// TwinCAT 3 PLC project Virtual_plc
// ProgramVersion: 3.1.4024.0
// libraries:
//   Tc2_Standard, * (Beckhoff Automation GmbH)
//   Tc2_System, * (Beckhoff Automation GmbH)
//   Tc3_Module, * (Beckhoff Automation GmbH)
// project tree:
//   GVLs/ GVL.TcGVL
//   / PlcTask.TcTTO, TASK_2.TcTTO
//   POUs/ Wait.TcPOU, Step.TcDUT, Task_1.TcPOU, Taks_2.TcPOU
// real-time tasks:
//   TASK PlcTask: cycle T#3000ms, priority 20, ADS port 350
//   TASK TASK 2: cycle T#1ms, priority 1, ADS port 351

CONFIGURATION Virtual_plc
    RESOURCE PLC ON TwinCAT3
        TASK PlcTask(INTERVAL := T#3000ms, PRIORITY := 20);
        TASK TASK_2(INTERVAL := T#1ms, PRIORITY := 1);
        PROGRAM Task_1 WITH PlcTask : Task_1;
        PROGRAM Taks_2 WITH TASK_2 : Taks_2;
    END_RESOURCE
END_CONFIGURATION

// ---- POUs/Step.TcDUT
TYPE Step :
//ALl the case steps
(
	sleeping, 
	alarm, 
	snooze1, 
	snooze2, 
	wake, 
	toilet1,
	kitchen, 
	breakfast, 
	lunch, 
	toilet2, 
	garage, 
	cycling,
	train_check, 
	done	
) := sleeping;
END_TYPE

// ---- GVLs/GVL.TcGVL
{attribute 'qualified_only'}
VAR_GLOBAL
    Delay : INT := 0;              // totale vertraging
	need_1 : INT := 10;
END_VAR

// ---- POUs/Task_1.TcPOU
// MAIN was replaced by EventTracker and DelayTracker
PROGRAM Task_1
VAR
	CurrentStep : step := sleeping;
    (* Alarm & Sleep *)
    AlarmSet          : BOOL := TRUE;
    Snooze1Wanted     : BOOL := TRUE;
    Snooze2Wanted     : BOOL := FALSE;
    StillTired        : BOOL := FALSE;

    (* Toilet choices *)
    ToiletMorning1    : BOOL := FALSE;
	geweest			:Bool := False;
    ToiletMorning2    : BOOL := FALSE;
	

    (* Breakfast *)
    StillHungry       : BOOL := TRUE;
    BreakfastCount    : INT := 0;

    (* Lunch *)
    MakeLunch         : BOOL := TRUE;
    WantSpeculoos     : BOOL := TRUE;
    WantChickenFilet  : BOOL := FALSE;
    WantPeanutButter  : BOOL := FALSE;

    SpeculoosAvail    : BOOL := TRUE;
    ChickenAvail      : BOOL := TRUE;
    PeanutAvail       : BOOL := TRUE;

    ToppingCount      : INT := 0;

    (* Cycling *)
    TrafficLightRed   : BOOL := TRUE;
    BridgeOpen        : BOOL := FALSE;

    (* Delay tracking *)
    DelayMinutes      : INT := 0;
    TrainDelayLimit   : INT := 10;
	Wait : Wait;
END_VAR

//Currentstep := sleeping;
IF gvl.need_1 > 50 THEN
	ToiletMorning1 := TRUE;
	ELSIF gvl.need_1 > 50 AND geweest = FALSE THEN
	ToiletMorning2 := TRUE;
END_IF




CASE CurrentStep OF

(* --------------------------- SLEEPING --------------------------- *)
sleeping:
    IF AlarmSet THEN
		Wait();
		IF wait.Klaar = TRUE THEN
			CurrentStep := alarm;
		END_IF    
    ELSE
        IF StillTired THEN
            GVL.Delay := GVL.Delay + 5;
			stillTired := FALSE;
        ELSE
			Wait();
			IF wait.Klaar = TRUE THEN
				CurrentStep := wake;
			END_IF
        END_IF
    END_IF

(* --------------------------- ALARM --------------------------- *)
alarm:
    IF Snooze1Wanted THEN
		Wait();
		IF wait.Klaar = TRUE THEN
			CurrentStep := snooze1;
		END_IF 
    ELSE
        CurrentStep := wake;
    END_IF

(* --------------------------- SNOOZE 1 --------------------------- *)
snooze1:
    DelayMinutes := DelayMinutes + 5;
    IF Snooze2Wanted THEN
	Wait();
	IF wait.Klaar = TRUE THEN
		CurrentStep := snooze2;
	END_IF 
    ELSE
        CurrentStep := wake;
    END_IF

(* --------------------------- SNOOZE 2 --------------------------- *)
snooze2:
    DelayMinutes := DelayMinutes + 5;
    CurrentStep := wake;

(* --------------------------- WAKE --------------------------- *)
wake:
    IF ToiletMorning1 THEN
        CurrentStep := toilet1;
    ELSE
        CurrentStep := kitchen;
    END_IF

(* --------------------------- FIRST TOILET --------------------------- *)
toilet1:
	IF ToiletMorning1 = TRUE THEN
		DelayMinutes := DelayMinutes + 2;
		gvl.need_1 := 0;
		geweest := TRUE;
		Wait();
		IF wait.Klaar = TRUE THEN
		CurrentStep := kitchen;
		END_IF
		ELSE
		CurrentStep := kitchen;
	END_IF
	
    
(* --------------------------- ENTER KITCHEN --------------------------- *)
kitchen:
    BreakfastCount := 0;
    CurrentStep := breakfast;

(* --------------------------- BREAKFAST LOOP --------------------------- *)
breakfast:
    IF StillHungry THEN
        BreakfastCount := BreakfastCount + 1;
        StillHungry := FALSE;
    ELSE
        CurrentStep := lunch;
    END_IF

(* --------------------------- LUNCH PREPARATION --------------------------- *)
lunch:
    IF MakeLunch THEN

        IF ToppingCount < 4 THEN

            IF WantSpeculoos THEN
                IF SpeculoosAvail THEN
                    ToppingCount := ToppingCount + 1;
                END_IF

            ELSIF WantChickenFilet THEN
                IF ChickenAvail THEN
                    ToppingCount := ToppingCount + 1;
                END_IF

            ELSIF WantPeanutButter THEN
                IF PeanutAvail THEN
                    ToppingCount := ToppingCount + 1;
                END_IF

            END_IF

        ELSE
            CurrentStep := toilet2; (* lunch packed *)
        END_IF

    ELSE
        CurrentStep := toilet2;
    END_IF

(* --------------------------- SECOND TOILET --------------------------- *)
toilet2:
    	IF ToiletMorning2 = TRUE THEN
		 DelayMinutes := DelayMinutes + 2;
		 gvl.need_1 := 0;
		Wait();
		IF wait.Klaar = TRUE THEN
		CurrentStep := garage;
		END_IF
		ELSE
		CurrentStep := garage;
	END_IF
(* --------------------------- GARAGE --------------------------- *)
garage:
	IF wait.Klaar = TRUE THEN
		CurrentStep := cycling;
	END_IF   

(* --------------------------- CYCLING --------------------------- *)
cycling:
    IF TrafficLightRed THEN
        DelayMinutes := DelayMinutes + 2;
    END_IF

    IF BridgeOpen THEN
        DelayMinutes := DelayMinutes + 5;
    END_IF

    CurrentStep := train_check;

(* --------------------------- TRAIN CHECK --------------------------- *)
train_check:
    IF DelayMinutes > TrainDelayLimit THEN
        (* Missed the train, but simulation ends here anyway *)
    END_IF

    CurrentStep := done;

(* --------------------------- DONE --------------------------- *)
done:
    (* Simulation finished *)
    ;

END_CASE

END_PROGRAM

// ---- POUs/Wait.TcPOU
FUNCTION_BLOCK Wait
VAR_OUTPUT
    Klaar : BOOL := FALSE;     // wordt TRUE na 5 seconden
END_VAR

VAR
    Tmr : TON;                 // interne timer
    Running : BOOL := FALSE;   // onthoudt of timer al gestart is
	flase: BOOL;
	done: BOOL;
	test: int;
END_VAR

// Timer automatisch starten zodra FB wordt opgeroepen
Tmr(IN := TRUE, PT := T#5S);
IF Done = TRUE THEN
klaar := FALSE;
tmr(IN := FALSE);
Done := FALSE;
END_IF
IF Tmr.Q THEN
	done := TRUE;
	klaar := TRUE;
END_IF

END_FUNCTION_BLOCK

// ---- POUs/Taks_2.TcPOU
PROGRAM Taks_2
VAR
	need: INT;
	timer: TON;	
	Wait5s: Wait;
END_VAR

//GVL.need_1 := 0;
IF GVL.need_1 < 100 THEN
	timer(IN := TRUE, PT := T#1S);
	IF timer.Q = TRUE THEN
		gvl.need_1 := gvl.need_1+1;	
		timer(IN := FALSE);
	END_IF
END_IF

END_PROGRAM
